// TIA Portal V20 export
FUNCTION "DemoIdentMv" : Void   // FC69, LAD
TITLE = Demo: Ident
AUTHOR : SICAR
FAMILY : Demo
VERSION : 1.0
// Demo for usage of ident moduls
// stored: IsIECCheckEnabled true, SetENOAutomatically true
   // Ret_Val : Ret_Val
BEGIN

REGION Network 1: ChangeLog
   // Change log table:
   // Version | Date | Expert in charge | Changes applied
   // -------|---------|-------------|--------------------------------------------
   // 05.00.00 | 01.09.2023 | SICAR | First released version
END_REGION

REGION Network 2: Call: Ident MV
   // Demonstrate the call and function of an optical reader MV device
END_REGION

REGION Network 3: Define reading informations
   // Write the String "Siemens" in the writting structur of the FB
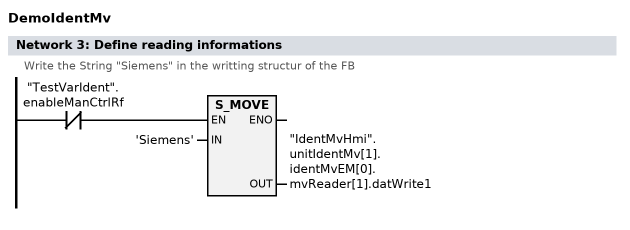
   RUNG wire#powerrail
      I_Contact( "TestVarIdent".enableManCtrlRf )
      S_Move(in := 'Siemens', out => "IdentMvHmi".unitIdentMv[1].identMvEM[0].mvReader[1].datWrite1)
   END_RUNG
   // the same network as SCL:
   IF NOT "TestVarIdent".enableManCtrlRf THEN
       "IdentMvHmi".unitIdentMv[1].identMvEM[0].mvReader[1].datWrite1 := 'Siemens';
   END_IF;
END_REGION
END_FUNCTION
